TYPE ST_ToolDataX :
STRUCT
	{attribute 'OPC.UA.DA.Description' := 'Job data type'}

END_STRUCT
END_TYPE

(* stored: Version 1.1.0.1, ProductVersion 3.1.4024.5
   DUT ST_ToolDataX: Id {e263d18d-ef7e-47dc-a80f-2337af4c74b1} *)
